(* Schneider Machine Expert - Basic project schneider, file version 2.7.0.0 *)
(* ProjectInformations: Name=New project *)

HARDWARE
  Cpu 0: TM200C24R
  EthernetConfiguration: NetworkName=M200, IpAllocationMode=FixedAddress, IpAddress=0.0.0.0, SubnetMask=0.0.0.0
  SerialLineConfiguration: Baud=Baud19200, Parity=ParityEven, DataBits=DataBits8, StopBits=StopBits1, PhysicalMedium=PhysicalMediumRs485, TransmissionMode=TransmissionModeModbusRtu, SlaveId=1, Addressing=SlaveAddressing
  MastTask: UsePeriodScanMode=false, PeriodScan=100
  FastTask: Period=255
  CpuBehavior: StartingMode=StartAsPreviousState, AutoSaveRamOnEeprom=true, WatchdogPeriod=250

SYMBOLS  (address, symbol, comment, settings)
  %TM0        [Preset=5, Base=OneSecond]
  %TM1        [Preset=5, Base=OneSecond]
  %TM2        [Preset=5, Base=OneSecond]

POU New POU
  (* SectionNumber=0 *)

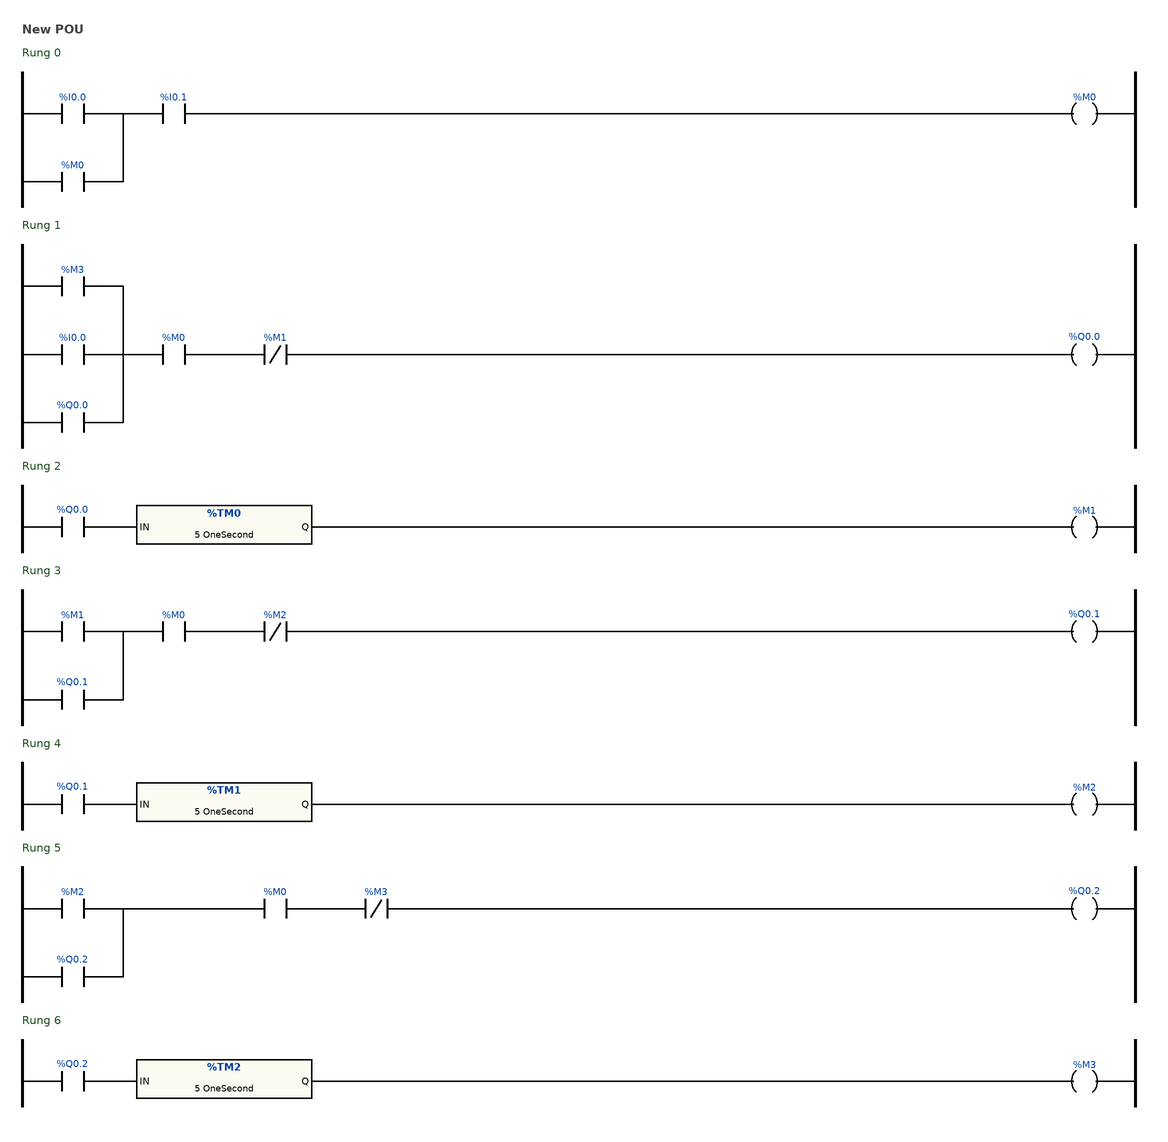

// Rung 0
  LD %I0.0
  OR %M0
  AND %I0.1
  ST %M0
  // as ST:
  //   %M0 := (%I0.0 OR %M0) AND %I0.1;

// Rung 1
  LD %M3
  OR %I0.0
  OR %Q0.0
  AND %M0
  ANDN %M1
  ST %Q0.0
  // as ST:
  //   %Q0.0 := (%M3 OR %I0.0 OR %Q0.0) AND %M0 AND NOT %M1;

// Rung 2
  BLK %TM0
  LD %Q0.0
  IN
  OUT_BLK
  LD Q
  ST %M1
  END_BLK
  // as ST:
  //   %TM0(IN := %Q0.0);
  //   %M1 := %TM0.Q;

// Rung 3
  LD %M1
  OR %Q0.1
  AND %M0
  ANDN %M2
  ST %Q0.1
  // as ST:
  //   %Q0.1 := (%M1 OR %Q0.1) AND %M0 AND NOT %M2;

// Rung 4
  BLK %TM1
  LD %Q0.1
  IN
  OUT_BLK
  LD Q
  ST %M2
  END_BLK
  // as ST:
  //   %TM1(IN := %Q0.1);
  //   %M2 := %TM1.Q;

// Rung 5
  LD %M2
  OR %Q0.2
  AND %M0
  ANDN %M3
  ST %Q0.2
  // as ST:
  //   %Q0.2 := (%M2 OR %Q0.2) AND %M0 AND NOT %M3;

// Rung 6
  BLK %TM2
  LD %Q0.2
  IN
  OUT_BLK
  LD Q
  ST %M3
  END_BLK
  // as ST:
  //   %TM2(IN := %Q0.2);
  //   %M3 := %TM2.Q;
